{attribute addProperty BoxType "AX8108-0000-0102-0102"}
{attribute addProperty Id "DeviceDevice_F82A60211620Ch_ACh_A_B17182A2176220WcStateAT %I*WcState_98A4DF7520.250InfoDataAT %I*InfoData_F030DC9B200250"}
{attribute addProperty CRC "3898025815"}
{attribute addProperty SizeInBites "394"}
{attribute addProperty SizeInBytes "49.25"}
TYPE AX8108_2B905711 :
STRUCT
	{attribute addProperty Name "Device"}
	Device : Device_F82A6021;
	{attribute addProperty Name "Ch_A"}
	Ch_A : Ch_A_B17182A2;
	{attribute addProperty Name "WcState"}
	WcState : WcState_98A4DF75;
	{attribute addProperty Name "InfoData"}
	InfoData : InfoData_F030DC9B;
END_STRUCT
END_TYPE

(* stored: Version 1.2.0.0, ProductVersion 3.1.4024.9
   DUT AX8108_2B905711: Id {6df35b1b-d514-49a1-a48f-8f2138fcf0e6} *)
